(* PLC project Main, Beckhoff Automation GmbH TwinCAT PLC Control 3.5.13.21 *)
(* stored: creationDateTime 2024-10-31T10:03:35.4772198, modificationDateTime 2024-10-31T10:03:35.4772198 *)

FUNCTION SinusFunction : REAL
VAR_INPUT
	A : 	REAL; 		//Amplitude
	yoff : 	REAL;		//Offset
	w : 	REAL;		//Kreisfrequenz
	t : 	REAL;		//Zeit
END_VAR
VAR
END_VAR

            SinusFunction := A * sin(w*t) + yoff;
RETURN;
          
END_FUNCTION
